// TIA Portal V19 export
FUNCTION "AnalogReadingSystem" : Void   // FC11, STL
TITLE = Analog Input Reading
{ S7_Optimized_Access := 'TRUE' }
AUTHOR : FLA
FAMILY : UHT
NAME : ANALO_IN
VERSION : 1.0
// Reads an analog input, scales it at transfers it to a word
// ------------------------------------------------------
// Programmer Init: 8953-FLA
// 
// Change Log:
// 
// Date        Change                          Updated by
// ------------------------------------------------------
// 01.03.99    1. Edition                      FLA
// stored: AutoNumber false
   VAR_INPUT
      IN_PIW : Word;
      MAX_REAL : Real;
      MIN_REAL : Real;
   END_VAR
   VAR_OUTPUT
      OUT_REAL : Real;
   END_VAR
   VAR_TEMP
      MAX_MIN : Real;
      IN_REAL : Real;
   END_VAR
BEGIN

NETWORK
TITLE = ANALO_IN
// Analog Input Reading
      L     #IN_PIW;
      ITD;
      DTR;
      T     #IN_REAL;
      L     #MAX_REAL;
      L     #MIN_REAL;
      -R;
      T     #MAX_MIN;
      L     #IN_REAL;
      L     #MAX_MIN;
      *R;
      L     27648.0;
      /R;
      L     #MIN_REAL;
      +R;
      T     #OUT_REAL;
END_FUNCTION
